INTERFACE I_Button EXTENDS I_Base

{attribute 'monitoring' := 'call'}
PROPERTY Active : BOOL
GET
END_GET
END_PROPERTY

{attribute 'monitoring' := 'call'}
PROPERTY Name : STRING
GET
END_GET
SET
END_SET
END_PROPERTY

PROPERTY Permissive : I_Permissive
GET
END_GET
END_PROPERTY

END_INTERFACE

(* stored: Version 1.1.0.1, ProductVersion 3.1.4026.18
   Itf I_Button: Id {dc87b376-9916-4af0-b5fb-3937dc1a1a2c}
   Property Active: Id {24e556cb-0ac4-4670-b3f5-d0f94d4c1f94}
   Get Get: Id {c0ce9bb1-7ab7-4676-a85d-a4e9df869101}
   Property Name: Id {5e539ec9-7038-4c4c-9689-84749789b947}
   Get Get: Id {f4ea3554-5f9f-49f0-8c57-003b2c39adbb}
   Set Set: Id {7d1ddbf2-6324-4d29-89f2-584b1e602a64}
   Property Permissive: Id {91674e1c-496e-4ecb-a243-af4070a47c12}
   Get Get: Id {ba58a541-451c-40f3-a2c6-430b9a3dc1c3} *)
